// TIA Portal V17 export
// export: Created 2024-01-30T08:49:13.3569546Z, ExportSetting WithDefaults, DisplayName Totally Integrated Automation Portal, DisplayVersion V17 Update 6, DisplayName TIA Portal Openness, DisplayVersion V17 Update 6, DisplayName TIA Portal Version Control Interface, DisplayVersion V17, DisplayName STEP 7 Professional, DisplayVersion V17 Update 6, DisplayName STEP 7 Safety, DisplayVersion V17 Update 6, DisplayName WinCC Advanced, DisplayVersion V17 Update 6
DATA_BLOCK "Keyence_LJX8000_CTRL_DB"   // DB27
VERSION : 0.1
// stored: AutoNumber true, DBAccessibleFromOPCUA true, DBAccessibleFromWebserver true, InstanceOfName Keyence_LJX8000_CTRL, InstanceOfType FB
"Keyence_LJX8000_CTRL"
   // VAR_INPUT
   //    PLC_IN_Bits : "UDT_LJ_X8000 --> PLC_Bits";
   //    PLC_IN_Bytes : "UDT_LJ_X8000 --> PLC_Bytes";
   //    RESET : Bool;
   //    CMD_NUMBER : DInt;
   //    PRG_NUMBER : DInt;
   //    CMD_REQ : Bool;
   //    TRIGGER : Bool;
   //    SD_CARD_NUM : DInt;
   // END_VAR
   // VAR_OUTPUT
   //    ERROR : Bool;
   //    ACTIVE_CMD : DInt;
   //    ACTIVE_PRG : DInt;
   //    CMD_READY : Bool;
   //    HEAD_READY : Bool;
   //    HEAD_BUSY : Bool;
   //    SYSTEM_RUN : Bool;
   //    CMD_COMPLETE : Bool;
   // END_VAR
   // VAR_IN_OUT
   //    PLC_OUT_Bits : "UDT_PLC --> LJ_X8000_Bits";
   //    PLC_Out_Bytes : "UDT_PLC --> LJ_X8000_Bytes";
   // END_VAR
   // VAR
   //    ChangeToRun : Bool;
   //    ChangeToSetup : Bool;
   // END_VAR
BEGIN
END_DATA_BLOCK
